FUNCTION_BLOCK C_HTTPSTREAM IMPLEMENTS I_STREAM
VAR_INPUT
END_VAR
VAR_OUTPUT
END_VAR
VAR
	_BASE_MEM : POINTER TO BYTE;
	_BASE_SIZE: UDINT;
	
	_STREAM_POSITION : UDINT := 0;
END_VAR

PROPERTY BufferSize : UDINT
GET
END_GET
END_PROPERTY

METHOD Close : DINT
VAR_INPUT
END_VAR
_BASE_MEM := 0;
_BASE_SIZE:= 0;
_STREAM_POSITION := 0;
Close := -1;
RETURN;
END_METHOD

PROPERTY EndOfStream : BOOL
GET
EndOfStream := _STREAM_POSITION >= _BASE_SIZE;
END_GET
END_PROPERTY

PROPERTY IsValid : BOOL
GET
IsValid := _BASE_MEM <> 0;
END_GET
END_PROPERTY

METHOD NEW : DINT
VAR_INPUT
	PTR_BASE	: PVOID;
	BASE_SIZE	: UDINT;
END_VAR
IF PTR_BASE = 0 OR BASE_SIZE = 0 OR IsValid THEN
	NEW := 1;
	RETURN;
ELSE
	_BASE_MEM := PTR_BASE;
	_BASE_SIZE:= BASE_SIZE;
	_STREAM_POSITION := 0;
	NEW := -1;
	RETURN;
END_IF
END_METHOD

METHOD Peek : DINT
VAR_INPUT
	ptr_DataOut : POINTER TO BYTE;
END_VAR
IF NOT IsValid THEN
	Peek := 1;
	RETURN;
END_IF

ptr_DataOut^ := _BASE_MEM[_STREAM_POSITION];
Peek := -1;
RETURN;
END_METHOD

PROPERTY Position : UDINT
GET
Position := _STREAM_POSITION;
END_GET
END_PROPERTY

METHOD Read : DINT
VAR_INPUT
	ptr_DataOut : PVOID;
	Length		: UDINT;
END_VAR
IF NOT IsValid THEN
	Read := 1;
	RETURN;
END_IF

IF _STREAM_POSITION + Length > _BASE_SIZE THEN
	Read := 2;
	RETURN;
END_IF
		
MEMCPY(ptr_DataOut, _BASE_MEM + _STREAM_POSITION, Length);
_STREAM_POSITION := _STREAM_POSITION + Length;
READ := -1;
RETURN;
END_METHOD

METHOD Seek : DINT
VAR_INPUT
	Offset 		: UDINT;
	SeekStyle 	: E_STREAMSEEKTYPE;
END_VAR
IF NOT IsValid THEN
	Seek := 1;
	RETURN;
END_IF

CASE SeekStyle OF
	E_STREAMSEEKTYPE.Current_Reversed:
		IF OFFSET > _STREAM_POSITION THEN
			Seek := 2;
			RETURN;
		ELSE
			_STREAM_POSITION := _STREAM_POSITION - OFFSET;
			Seek := -1;
			RETURN;
		END_IF
	E_STREAMSEEKTYPE.Current:
		IF _STREAM_POSITION + OFFSET >= _BASE_SIZE THEN
			Seek := 2;
			RETURN;
		ELSE
			_STREAM_POSITION := _STREAM_POSITION + OFFSET;
			Seek := -1;
			RETURN;
		END_IF
	E_STREAMSEEKTYPE.End:
		IF OFFSET >= _BASE_SIZE THEN
			Seek := 2;
			RETURN;
		ELSE
			_STREAM_POSITION := _BASE_SIZE - Offset - 1;
			Seek := -1;
			RETURN;
		END_IF
	E_STREAMSEEKTYPE.Origin:
		IF OFFSET >= _BASE_SIZE THEN
			Seek := 2;
			RETURN;
		ELSE
			_STREAM_POSITION := Offset;
			Seek := -1;
			RETURN;
		END_IF
END_CASE
END_METHOD

METHOD Write : DINT
VAR_INPUT
	ptr_DataIn	: PVOID;
	Length		: UDINT;
END_VAR
IF NOT IsValid THEN
	Write := 1;
	RETURN;
END_IF

IF _STREAM_POSITION + Length > _BASE_SIZE THEN
	Write := 2;
	RETURN;
END_IF
		
MEMCPY(_BASE_MEM + _STREAM_POSITION, ptr_DataIn, Length);
_STREAM_POSITION := _STREAM_POSITION + Length;
Write := -1;
RETURN;
END_METHOD

END_FUNCTION_BLOCK

(* stored: Version 1.1.0.1, ProductVersion 3.1.4020.3
   POU C_HTTPSTREAM: Id {60f91825-763a-47ae-92e4-2306c3d57054}, SpecialFunc None
   Folder Methods: Id {729a20d3-cfb4-4999-9424-e1f47fd1662f}
   Folder Properties: Id {24196728-f538-4a63-824a-61e753046204}
   Property BufferSize: Id {dcf112fc-2290-4f03-81fd-e0797dd1c536}
   Get Get: Id {46208aba-2fbe-459e-ac17-ad0df3e2c76c}
   Method Close: Id {7c44b1b5-1c79-4683-af1b-6f22a4dd7ab2}
   Property EndOfStream: Id {28bb4416-fc2a-42fb-8e1a-c4bf281661c6}
   Get Get: Id {0a2a77ff-c247-4c90-87e2-957556706494}
   Property IsValid: Id {5c18e574-f6c3-4efa-901a-ad689c4f1e96}
   Get Get: Id {23e44237-8493-481d-aa87-9d898e09bc4b}
   Method NEW: Id {44cdb0df-6e4c-4ffc-a15d-ecd6e8eb792a}
   Method Peek: Id {e16edd05-f2c4-473e-ab91-2b575e73de6f}
   Property Position: Id {6d955390-abde-48c4-b867-2bf6eaa7ff00}
   Get Get: Id {a43296ce-00a7-464b-9e99-aed0a73e4f2c}
   Method Read: Id {0fd092b8-6a3f-4e32-a482-13b517200186}
   Method Seek: Id {88daf200-5ac7-40da-9e52-e8daa23386b3}
   Method Write: Id {7008c3e7-909a-4d23-9ec1-6df3be7e9a28} *)
